# EPICS substitutions: db/core/ecmcPlc.substitutions
file ecmcPlc.template
{
  pattern { PLC_ENABLE,               PLC_SCANTIME,               PLC_ERROR,            DESC_NAME}
          { PLC$(Index2Char)-EnaCmd,  PLC$(Index2Char)-ScanTime,  PLC$(Index2Char)-Err, PLC$(Index2Char)-Desc }
}
